ABB RAPID module: StanTargets.mod

MODULE StanTargets

	!Workplan Variables
	CONST string workplanName := "Stan";
	CONST string workplanUUID := "d4fdb9e9-5a3f-4a80-8776-aeeac0a44db1";

	!Workingsteps
	CONST string WorkPlan{20,6} := [
		["1","7", "Drilling.2", "b062b09d-c75e-4509-b058-f533fc3121cb", "Hole.101", "7ba2387a-5122-471d-9e62-f4dd978dd916"],
		["8","14", "Drilling.19", "bc6d7e2e-2011-44a2-96ea-1bdf43305bb2", "Hole.2", "a5a2d4b3-bce9-4376-9a01-39ac46aa03b7"],
		["15","21", "Drilling.20", "1d99434e-626c-49cd-aa28-89c40de30f06", "Hole.105", "77f1627f-4d66-488f-b970-3b2b6af52deb"],
		["22","28", "Drilling.3", "45a28ad3-0738-4ba8-bc95-27ca5d3c2a9d", "Hole.102", "83a55789-a548-457f-bc7a-c5f73e279b59"],
		["29","35", "Drilling.1", "9e701cf1-a52e-421d-a5d1-a7fe2dbaa640", "Hole.100", "ec9e4cb9-16a2-432e-8136-2d658a3c3d31"],
		["36","42", "Drilling.18", "90b44a9d-16c4-4a88-bf09-b7f65aff8308", "Hole.106", "8309f7bd-9ba6-4400-9e0b-e392acc79543"],
		["43","49", "Drilling.4", "301b61b0-be88-4471-af20-9d54f270abc0", "Hole.103", "543c12c8-ac8b-46e2-b23c-ed2f3937359b"],
		["50","56", "Drilling.17", "4a6a49de-cb15-4803-8bb7-097c767e5d1a", "Hole.107", "bc5d4dfc-6aa2-4544-8bb1-6cd32004e75e"],
		["57","63", "Drilling.21", "d6a29b26-5ed6-4fc9-a609-95bc5c10512a", "Hole.109", "c5793a88-d117-412a-8380-89480e2aa149"],
		["64","70", "Drilling.22", "32b13ef1-a017-413c-926d-f3ce9280a815", "Hole.110", "f43400ad-c29f-4157-ba87-1fd86718dbb4"],
		["71","77", "Drilling.23", "961958d8-0134-4891-910a-03c3b0fd50ac", "Hole.111", "4c4ae24f-0e25-46c1-affc-8b190d84e835"],
		["78","84", "Drilling.24", "46b8f9da-afaf-476f-bebf-76b29446400a", "Hole.112", "58a054b0-4018-4bcc-8be0-6224a9ae077a"],
		["85","91", "Drilling.37", "a26de890-fc0a-49b5-bfdf-50d0ba577d7f", "Hole.117", "fd2c949e-3c41-489a-8a46-dd0d10567b1b"],
		["92","98", "Drilling.38", "57e6c193-12b5-426e-af89-bc1afa04e779", "Hole.116", "13521d27-8989-4ee6-aa90-747ab0996569"],
		["99","105", "Drilling.39", "43fec44c-5451-4481-a3ed-f2154e5b5857", "Hole.115", "b8ea09e7-7ee5-4781-9867-97bdf0c7c8c2"],
		["106","112", "Drilling.40", "b2407ed9-3760-41ef-9af3-e4b017b94bad", "Hole.114", "6fd1afc0-306a-4e0e-985a-70eb87f380a3"],
		["113","119", "Drilling.41", "e4391847-02d9-4746-a9c4-e995e37bf0a5", "Hole.119", "2fe5694b-30b9-4983-885c-0907e4daf0a7"],
		["120","126", "Drilling.42", "9648c8b5-7603-4606-8e84-4fa243c23e6f", "Hole.120", "7e69786d-15ab-4ddf-bc4f-041c788858b9"],
		["127","133", "Drilling.43", "1797812d-a7bf-4001-89eb-f8bf3d30d00a", "Hole.121", "a39c1e68-904f-4878-9c68-b76c3ab1c433"],
		["134","140", "Drilling.44", "c9657693-5bc7-40ba-995c-70b253dd4bce", "Hole.122", "35b9f3e4-dbe9-4a3b-b0cd-96909b64c764"]
		];

	!Positions
	CONST robtarget WorkingstepRobtargets{140} := [
		[[289.186156636195,-206.403560128169,35.3771625636731],[0.00835255338347923,-0.000732758938354189,-0.996138888459216,-0.0873900040940131],[0,0,0,0],[9E+09,9E+09,9E+09,9E+09,9E+09,9E+09]],
		[[288.347319864636,-197.55839601017,-14.6398287952277],[0.00835255338347923,-0.000732758938354189,-0.996138888459216,-0.0873900040940131],[0,0,0,0],[9E+09,9E+09,9E+09,9E+09,9E+09,9E+09]],
		[[288.347319864636,-197.55839601017,-14.6398287952277],[0.00835255338347923,-0.000732758938354189,-0.996138888459216,-0.0873900040940131],[0,0,0,0],[9E+09,9E+09,9E+09,9E+09,9E+09,9E+09]],
		[[287.823046882412,-192.030168436421,-45.9004483945406],[0.00835255338347923,-0.000732758938354189,-0.996138888459216,-0.0873900040940131],[0,0,0,0],[9E+09,9E+09,9E+09,9E+09,9E+09,9E+09]],
		[[287.823046882412,-192.030168436421,-45.9004483945406],[0.00835255338347923,-0.000732758938354189,-0.996138888459216,-0.0873900040940131],[0,0,0,0],[9E+09,9E+09,9E+09,9E+09,9E+09,9E+09]],
		[[288.347319864636,-197.55839601017,-14.6398287952277],[0.00835255338347923,-0.000732758938354189,-0.996138888459216,-0.0873900040940131],[0,0,0,0],[9E+09,9E+09,9E+09,9E+09,9E+09,9E+09]],
		[[289.186156636195,-206.403560128169,35.3771625636731],[0.00835255338347923,-0.000732758938354189,-0.996138888459216,-0.0873900040940131],[0,0,0,0],[9E+09,9E+09,9E+09,9E+09,9E+09,9E+09]],
		[[254.909208192728,-190.980764818536,38.5531834909307],[0.00803255668836741,-0.000646350507138514,-0.996745854533864,-0.0802044994599877],[0,0,0,0],[9E+09,9E+09,9E+09,9E+09,9E+09,9E+09]],
		[[254.101023132797,-182.857977487938,-11.5866924850904],[0.00803255668836741,-0.000646350507138514,-0.996745854533864,-0.0802044994599877],[0,0,0,0],[9E+09,9E+09,9E+09,9E+09,9E+09,9E+09]],
		[[254.101023132797,-182.857977487938,-11.5866924850904],[0.00803255668836741,-0.000646350507138514,-0.996745854533864,-0.0802044994599877],[0,0,0,0],[9E+09,9E+09,9E+09,9E+09,9E+09,9E+09]],
		[[253.595907470339,-177.781235406315,-42.9241149701038],[0.00803255668836741,-0.000646350507138514,-0.996745854533864,-0.0802044994599877],[0,0,0,0],[9E+09,9E+09,9E+09,9E+09,9E+09,9E+09]],
		[[253.595907470339,-177.781235406315,-42.9241149701038],[0.00803255668836741,-0.000646350507138514,-0.996745854533864,-0.0802044994599877],[0,0,0,0],[9E+09,9E+09,9E+09,9E+09,9E+09,9E+09]],
		[[254.101023132797,-182.857977487938,-11.5866924850904],[0.00803255668836741,-0.000646350507138514,-0.996745854533864,-0.0802044994599877],[0,0,0,0],[9E+09,9E+09,9E+09,9E+09,9E+09,9E+09]],
		[[254.909208192728,-190.980764818536,38.5531834909307],[0.00803255668836741,-0.000646350507138514,-0.996745854533864,-0.0802044994599877],[0,0,0,0],[9E+09,9E+09,9E+09,9E+09,9E+09,9E+09]],
		[[255.049346094491,-251.794133959213,27.0746013914174],[0.00931771731230624,-0.000993284320775785,-0.994322356952738,-0.105996433875385],[0,0,0,0],[9E+09,9E+09,9E+09,9E+09,9E+09,9E+09]],
		[[254.118737842067,-241.085099842443,-22.5750769214012],[0.00931771731230624,-0.000993284320775785,-0.994322356952738,-0.105996433875385],[0,0,0,0],[9E+09,9E+09,9E+09,9E+09,9E+09,9E+09]],
		[[254.118737842067,-241.085099842443,-22.5750769214012],[0.00931771731230624,-0.000993284320775785,-0.994322356952738,-0.105996433875385],[0,0,0,0],[9E+09,9E+09,9E+09,9E+09,9E+09,9E+09]],
		[[253.5371076843,-234.391953519461,-53.6061258669128],[0.00931771731230624,-0.000993284320775785,-0.994322356952738,-0.105996433875385],[0,0,0,0],[9E+09,9E+09,9E+09,9E+09,9E+09,9E+09]],
		[[253.5371076843,-234.391953519461,-53.6061258669128],[0.00931771731230624,-0.000993284320775785,-0.994322356952738,-0.105996433875385],[0,0,0,0],[9E+09,9E+09,9E+09,9E+09,9E+09,9E+09]],
		[[254.118737842067,-241.085099842443,-22.5750769214012],[0.00931771731230624,-0.000993284320775785,-0.994322356952738,-0.105996433875385],[0,0,0,0],[9E+09,9E+09,9E+09,9E+09,9E+09,9E+09]],
		[[255.049346094491,-251.794133959213,27.0746013914174],[0.00931771731230624,-0.000993284320775785,-0.994322356952738,-0.105996433875385],[0,0,0,0],[9E+09,9E+09,9E+09,9E+09,9E+09,9E+09]],
		[[288.817292795415,-151.336810998548,43.7919561194079],[0.00741254609803812,-0.000475090293762373,-0.997924837913392,-0.0639597242417948],[0,0,0,0],[9E+09,9E+09,9E+09,9E+09,9E+09,9E+09]],
		[[288.068828229942,-144.851630260459,-6.58683139665437],[0.00741254609803812,-0.000475090293762373,-0.997924837913392,-0.0639597242417948],[0,0,0,0],[9E+09,9E+09,9E+09,9E+09,9E+09,9E+09]],
		[[288.068828229942,-144.851630260459,-6.58683139665437],[0.00741254609803812,-0.000475090293762373,-0.997924837913392,-0.0639597242417948],[0,0,0,0],[9E+09,9E+09,9E+09,9E+09,9E+09,9E+09]],
		[[287.60103787652,-140.798392299153,-38.0735735941933],[0.00741254609803812,-0.000475090293762373,-0.997924837913392,-0.0639597242417948],[0,0,0,0],[9E+09,9E+09,9E+09,9E+09,9E+09,9E+09]],
		[[287.60103787652,-140.798392299153,-38.0735735941933],[0.00741254609803812,-0.000475090293762373,-0.997924837913392,-0.0639597242417948],[0,0,0,0],[9E+09,9E+09,9E+09,9E+09,9E+09,9E+09]],
		[[288.068828229942,-144.851630260459,-6.58683139665437],[0.00741254609803812,-0.000475090293762373,-0.997924837913392,-0.0639597242417948],[0,0,0,0],[9E+09,9E+09,9E+09,9E+09,9E+09,9E+09]],
		[[288.817292795415,-151.336810998548,43.7919561194079],[0.00741254609803812,-0.000475090293762373,-0.997924837913392,-0.0639597242417948],[0,0,0,0],[9E+09,9E+09,9E+09,9E+09,9E+09,9E+09]],
		[[293.28700751171,-244.361649311658,27.9483297927613],[0.00918827288987244,-0.000958205797942005,-0.994563756282914,-0.103718813005981],[0,0,0,0],[9E+09,9E+09,9E+09,9E+09,9E+09,9E+09]],
		[[292.368651285828,-233.880209617552,-21.7501213277837],[0.00918827288987244,-0.000958205797942005,-0.994563756282914,-0.103718813005981],[0,0,0,0],[9E+09,9E+09,9E+09,9E+09,9E+09,9E+09]],
		[[292.368651285828,-233.880209617552,-21.7501213277837],[0.00918827288987244,-0.000958205797942005,-0.994563756282914,-0.103718813005981],[0,0,0,0],[9E+09,9E+09,9E+09,9E+09,9E+09,9E+09]],
		[[291.794678644652,-227.329309808736,-52.8116532781243],[0.00918827288987244,-0.000958205797942005,-0.994563756282914,-0.103718813005981],[0,0,0,0],[9E+09,9E+09,9E+09,9E+09,9E+09,9E+09]],
		[[291.794678644652,-227.329309808736,-52.8116532781243],[0.00918827288987244,-0.000958205797942005,-0.994563756282914,-0.103718813005981],[0,0,0,0],[9E+09,9E+09,9E+09,9E+09,9E+09,9E+09]],
		[[292.368651285828,-233.880209617552,-21.7501213277837],[0.00918827288987244,-0.000958205797942005,-0.994563756282914,-0.103718813005981],[0,0,0,0],[9E+09,9E+09,9E+09,9E+09,9E+09,9E+09]],
		[[293.28700751171,-244.361649311658,27.9483297927613],[0.00918827288987244,-0.000958205797942005,-0.994563756282914,-0.103718813005981],[0,0,0,0],[9E+09,9E+09,9E+09,9E+09,9E+09,9E+09]],
		[[249.459094617476,-137.316682571751,46.0807019976294],[0.00720641123076419,-0.000415118187492874,-0.998318997016837,-0.0575071778942388],[0,0,0,0],[9E+09,9E+09,9E+09,9E+09,9E+09,9E+09]],
		[[248.730579441892,-131.483471005379,-4.37802280255641],[0.00720641123076419,-0.000415118187492874,-0.998318997016837,-0.0575071778942388],[0,0,0,0],[9E+09,9E+09,9E+09,9E+09,9E+09,9E+09]],
		[[248.730579441892,-131.483471005379,-4.37802280255641],[0.00720641123076419,-0.000415118187492874,-0.998318997016837,-0.0575071778942388],[0,0,0,0],[9E+09,9E+09,9E+09,9E+09,9E+09,9E+09]],
		[[248.275257457153,-127.837713776397,-35.9147258026727],[0.00720641123076419,-0.000415118187492874,-0.998318997016837,-0.0575071778942388],[0,0,0,0],[9E+09,9E+09,9E+09,9E+09,9E+09,9E+09]],
		[[248.275257457153,-127.837713776397,-35.9147258026727],[0.00720641123076419,-0.000415118187492874,-0.998318997016837,-0.0575071778942388],[0,0,0,0],[9E+09,9E+09,9E+09,9E+09,9E+09,9E+09]],
		[[248.730579441892,-131.483471005379,-4.37802280255641],[0.00720641123076419,-0.000415118187492874,-0.998318997016837,-0.0575071778942388],[0,0,0,0],[9E+09,9E+09,9E+09,9E+09,9E+09,9E+09]],
		[[249.459094617476,-137.316682571751,46.0807019976294],[0.00720641123076419,-0.000415118187492874,-0.998318997016837,-0.0575071778942388],[0,0,0,0],[9E+09,9E+09,9E+09,9E+09,9E+09,9E+09]],
		[[290.829543745998,-100.056182181525,49.234722450473],[0.00680707504627507,-0.000287946923608445,-0.999083317268074,-0.042262346982922],[0,0,0,0],[9E+09,9E+09,9E+09,9E+09,9E+09,9E+09]],
		[[290.139815300174,-95.7660646865366,-1.37910141761904],[0.00680707504627507,-0.000287946923608445,-0.999083317268074,-0.042262346982922],[0,0,0,0],[9E+09,9E+09,9E+09,9E+09,9E+09,9E+09]],
		[[290.139815300174,-95.7660646865366,-1.37910141761904],[0.00680707504627507,-0.000287946923608445,-0.999083317268074,-0.042262346982922],[0,0,0,0],[9E+09,9E+09,9E+09,9E+09,9E+09,9E+09]],
		[[289.708735021536,-93.0847412521693,-33.0127413351765],[0.00680707504627507,-0.000287946923608445,-0.999083317268074,-0.042262346982922],[0,0,0,0],[9E+09,9E+09,9E+09,9E+09,9E+09,9E+09]],
		[[289.708735021536,-93.0847412521693,-33.0127413351765],[0.00680707504627507,-0.000287946923608445,-0.999083317268074,-0.042262346982922],[0,0,0,0],[9E+09,9E+09,9E+09,9E+09,9E+09,9E+09]],
		[[290.139815300174,-95.7660646865366,-1.37910141761904],[0.00680707504627507,-0.000287946923608445,-0.999083317268074,-0.042262346982922],[0,0,0,0],[9E+09,9E+09,9E+09,9E+09,9E+09,9E+09]],
		[[290.829543745998,-100.056182181525,49.234722450473],[0.00680707504627507,-0.000287946923608445,-0.999083317268074,-0.042262346982922],[0,0,0,0],[9E+09,9E+09,9E+09,9E+09,9E+09,9E+09]],
		[[245.740187119161,-87.6128069534354,50.8276032034953],[0.0066909782554097,-0.000245268224154555,-0.999306424862602,-0.0366311326852939],[0,0,0,0],[9E+09,9E+09,9E+09,9E+09,9E+09,9E+09]],
		[[245.061768043552,-83.8934984330366,0.16848268519243],[0.0066909782554097,-0.000245268224154555,-0.999306424862602,-0.0366311326852939],[0,0,0,0],[9E+09,9E+09,9E+09,9E+09,9E+09,9E+09]],
		[[245.061768043552,-83.8934984330366,0.16848268519243],[0.0066909782554097,-0.000245268224154555,-0.999306424862602,-0.0366311326852939],[0,0,0,0],[9E+09,9E+09,9E+09,9E+09,9E+09,9E+09]],
		[[244.637756121297,-81.5689306077871,-31.493467638747],[0.0066909782554097,-0.000245268224154555,-0.999306424862602,-0.0366311326852939],[0,0,0,0],[9E+09,9E+09,9E+09,9E+09,9E+09,9E+09]],
		[[244.637756121297,-81.5689306077871,-31.493467638747],[0.0066909782554097,-0.000245268224154555,-0.999306424862602,-0.0366311326852939],[0,0,0,0],[9E+09,9E+09,9E+09,9E+09,9E+09,9E+09]],
		[[245.061768043552,-83.8934984330366,0.16848268519243],[0.0066909782554097,-0.000245268224154555,-0.999306424862602,-0.0366311326852939],[0,0,0,0],[9E+09,9E+09,9E+09,9E+09,9E+09,9E+09]],
		[[245.740187119161,-87.6128069534354,50.8276032034953],[0.0066909782554097,-0.000245268224154555,-0.999306424862602,-0.0366311326852939],[0,0,0,0],[9E+09,9E+09,9E+09,9E+09,9E+09,9E+09]],
		[[403.099233829671,-245.749127372575,25.6017542319324],[0.00936954043940217,-0.00100794170503457,-0.994219250722917,-0.106954556973674],[0,0,0,0],[9E+09,9E+09,9E+09,9E+09,9E+09,9E+09]],
		[[402.163744360367,-234.944401870427,-24.0270959086467],[0.00936954043940217,-0.00100794170503457,-0.994219250722917,-0.106954556973674],[0,0,0,0],[9E+09,9E+09,9E+09,9E+09,9E+09,9E+09]],
		[[402.163744360367,-234.944401870427,-24.0270959086467],[0.00936954043940217,-0.00100794170503457,-0.994219250722917,-0.106954556973674],[0,0,0,0],[9E+09,9E+09,9E+09,9E+09,9E+09,9E+09]],
		[[401.579063442052,-228.191448431585,-55.0451272465088],[0.00936954043940217,-0.00100794170503457,-0.994219250722917,-0.106954556973674],[0,0,0,0],[9E+09,9E+09,9E+09,9E+09,9E+09,9E+09]],
		[[401.579063442052,-228.191448431585,-55.0451272465088],[0.00936954043940217,-0.00100794170503457,-0.994219250722917,-0.106954556973674],[0,0,0,0],[9E+09,9E+09,9E+09,9E+09,9E+09,9E+09]],
		[[402.163744360367,-234.944401870427,-24.0270959086467],[0.00936954043940217,-0.00100794170503457,-0.994219250722917,-0.106954556973674],[0,0,0,0],[9E+09,9E+09,9E+09,9E+09,9E+09,9E+09]],
		[[403.099233829671,-245.749127372575,25.6017542319324],[0.00936954043940217,-0.00100794170503457,-0.994219250722917,-0.106954556973674],[0,0,0,0],[9E+09,9E+09,9E+09,9E+09,9E+09,9E+09]],
		[[396.033748937128,-194.18703812988,35.7216135201404],[0.00820516010917249,-0.000693329099167655,-0.996415168384063,-0.0841962401565701],[0,0,0,0],[9E+09,9E+09,9E+09,9E+09,9E+09,9E+09]],
		[[395.209024115822,-185.662788001459,-14.3513031985533],[0.00820516010917249,-0.000693329099167655,-0.996415168384063,-0.0841962401565701],[0,0,0,0],[9E+09,9E+09,9E+09,9E+09,9E+09,9E+09]],
		[[395.209024115822,-185.662788001459,-14.3513031985533],[0.00820516010917249,-0.000693329099167655,-0.996415168384063,-0.0841962401565701],[0,0,0,0],[9E+09,9E+09,9E+09,9E+09,9E+09,9E+09]],
		[[394.693571102503,-180.335131671196,-45.6468761477369],[0.00820516010917249,-0.000693329099167655,-0.996415168384063,-0.0841962401565701],[0,0,0,0],[9E+09,9E+09,9E+09,9E+09,9E+09,9E+09]],
		[[394.693571102503,-180.335131671196,-45.6468761477369],[0.00820516010917249,-0.000693329099167655,-0.996415168384063,-0.0841962401565701],[0,0,0,0],[9E+09,9E+09,9E+09,9E+09,9E+09,9E+09]],
		[[395.209024115822,-185.662788001459,-14.3513031985533],[0.00820516010917249,-0.000693329099167655,-0.996415168384063,-0.0841962401565701],[0,0,0,0],[9E+09,9E+09,9E+09,9E+09,9E+09,9E+09]],
		[[396.033748937128,-194.18703812988,35.7216135201404],[0.00820516010917249,-0.000693329099167655,-0.996415168384063,-0.0841962401565701],[0,0,0,0],[9E+09,9E+09,9E+09,9E+09,9E+09,9E+09]],
		[[391.06989532529,-137.544241837855,44.000996564666],[0.00726571628808549,-0.000432828028158066,-0.998203897421597,-0.0594642850714026],[0,0,0,0],[9E+09,9E+09,9E+09,9E+09,9E+09,9E+09]],
		[[390.335639388971,-131.51320224425,-6.43438218517918],[0.00726571628808549,-0.000432828028158066,-0.998203897421597,-0.0594642850714026],[0,0,0,0],[9E+09,9E+09,9E+09,9E+09,9E+09,9E+09]],
		[[390.335639388971,-131.51320224425,-6.43438218517918],[0.00726571628808549,-0.000432828028158066,-0.998203897421597,-0.0594642850714026],[0,0,0,0],[9E+09,9E+09,9E+09,9E+09,9E+09,9E+09]],
		[[389.876729428771,-127.743802498246,-37.9564939038324],[0.00726571628808549,-0.000432828028158066,-0.998203897421597,-0.0594642850714026],[0,0,0,0],[9E+09,9E+09,9E+09,9E+09,9E+09,9E+09]],
		[[389.876729428771,-127.743802498246,-37.9564939038324],[0.00726571628808549,-0.000432828028158066,-0.998203897421597,-0.0594642850714026],[0,0,0,0],[9E+09,9E+09,9E+09,9E+09,9E+09,9E+09]],
		[[390.335639388971,-131.51320224425,-6.43438218517918],[0.00726571628808549,-0.000432828028158066,-0.998203897421597,-0.0594642850714026],[0,0,0,0],[9E+09,9E+09,9E+09,9E+09,9E+09,9E+09]],
		[[391.06989532529,-137.544241837855,44.000996564666],[0.00726571628808549,-0.000432828028158066,-0.998203897421597,-0.0594642850714026],[0,0,0,0],[9E+09,9E+09,9E+09,9E+09,9E+09,9E+09]],
		[[385.668546901666,-85.4729115296458,49.1107245728777],[0.00669526575096486,-0.000247046366600005,-0.999297509827073,-0.0368727438364299],[0,0,0,0],[9E+09,9E+09,9E+09,9E+09,9E+09,9E+09]],
		[[384.989711265164,-81.7291044236946,-1.54658576365773],[0.00669526575096486,-0.000247046366600005,-0.999297509827073,-0.0368727438364299],[0,0,0,0],[9E+09,9E+09,9E+09,9E+09,9E+09,9E+09]],
		[[384.989711265164,-81.7291044236946,-1.54658576365773],[0.00669526575096486,-0.000247046366600005,-0.999297509827073,-0.0368727438364299],[0,0,0,0],[9E+09,9E+09,9E+09,9E+09,9E+09,9E+09]],
		[[384.565438992351,-79.389224982475,-33.2074047239924],[0.00669526575096486,-0.000247046366600005,-0.999297509827073,-0.0368727438364299],[0,0,0,0],[9E+09,9E+09,9E+09,9E+09,9E+09,9E+09]],
		[[384.565438992351,-79.389224982475,-33.2074047239924],[0.00669526575096486,-0.000247046366600005,-0.999297509827073,-0.0368727438364299],[0,0,0,0],[9E+09,9E+09,9E+09,9E+09,9E+09,9E+09]],
		[[384.989711265164,-81.7291044236946,-1.54658576365773],[0.00669526575096486,-0.000247046366600005,-0.999297509827073,-0.0368727438364299],[0,0,0,0],[9E+09,9E+09,9E+09,9E+09,9E+09,9E+09]],
		[[385.668546901666,-85.4729115296458,49.1107245728777],[0.00669526575096486,-0.000247046366600005,-0.999297509827073,-0.0368727438364299],[0,0,0,0],[9E+09,9E+09,9E+09,9E+09,9E+09,9E+09]],
		[[478.315791276222,-86.4437658870823,47.794069485851],[0.00671892774812616,-0.000256146261682229,-0.999251517650421,-0.038094551740885],[0,0,0,0],[9E+09,9E+09,9E+09,9E+09,9E+09,9E+09]],
		[[477.634650553439,-82.5760815046593,-2.85390248572684],[0.00671892774812616,-0.000256146261682229,-0.999251517650421,-0.038094551740885],[0,0,0,0],[9E+09,9E+09,9E+09,9E+09,9E+09,9E+09]],
		[[477.634650553439,-82.5760815046593,-2.85390248572684],[0.00671892774812616,-0.000256146261682229,-0.999251517650421,-0.038094551740885],[0,0,0,0],[9E+09,9E+09,9E+09,9E+09,9E+09,9E+09]],
		[[477.208937601699,-80.1587787656448,-34.5088849679627],[0.00671892774812616,-0.000256146261682229,-0.999251517650421,-0.038094551740885],[0,0,0,0],[9E+09,9E+09,9E+09,9E+09,9E+09,9E+09]],
		[[477.208937601699,-80.1587787656448,-34.5088849679627],[0.00671892774812616,-0.000256146261682229,-0.999251517650421,-0.038094551740885],[0,0,0,0],[9E+09,9E+09,9E+09,9E+09,9E+09,9E+09]],
		[[477.634650553439,-82.5760815046593,-2.85390248572684],[0.00671892774812616,-0.000256146261682229,-0.999251517650421,-0.038094551740885],[0,0,0,0],[9E+09,9E+09,9E+09,9E+09,9E+09,9E+09]],
		[[478.315791276222,-86.4437658870823,47.794069485851],[0.00671892774812616,-0.000256146261682229,-0.999251517650421,-0.038094551740885],[0,0,0,0],[9E+09,9E+09,9E+09,9E+09,9E+09,9E+09]],
		[[483.133106013849,-138.756801668918,42.5082331765351],[0.0073226084519266,-0.000449565472182051,-0.998093827794076,-0.0612771426856401],[0,0,0,0],[9E+09,9E+09,9E+09,9E+09,9E+09,9E+09]],
		[[482.393346029146,-132.54257687196,-7.904822328343],[0.0073226084519266,-0.000449565472182051,-0.998093827794076,-0.0612771426856401],[0,0,0,0],[9E+09,9E+09,9E+09,9E+09,9E+09,9E+09]],
		[[482.393346029146,-132.54257687196,-7.904822328343],[0.0073226084519266,-0.000449565472182051,-0.998093827794076,-0.0612771426856401],[0,0,0,0],[9E+09,9E+09,9E+09,9E+09,9E+09,9E+09]],
		[[481.930996038707,-128.658686373861,-39.4129820188915],[0.0073226084519266,-0.000449565472182051,-0.998093827794076,-0.0612771426856401],[0,0,0,0],[9E+09,9E+09,9E+09,9E+09,9E+09,9E+09]],
		[[481.930996038707,-128.658686373861,-39.4129820188915],[0.0073226084519266,-0.000449565472182051,-0.998093827794076,-0.0612771426856401],[0,0,0,0],[9E+09,9E+09,9E+09,9E+09,9E+09,9E+09]],
		[[482.393346029146,-132.54257687196,-7.904822328343],[0.0073226084519266,-0.000449565472182051,-0.998093827794076,-0.0612771426856401],[0,0,0,0],[9E+09,9E+09,9E+09,9E+09,9E+09,9E+09]],
		[[483.133106013849,-138.756801668918,42.5082331765351],[0.0073226084519266,-0.000449565472182051,-0.998093827794076,-0.0612771426856401],[0,0,0,0],[9E+09,9E+09,9E+09,9E+09,9E+09,9E+09]],
		[[483.222642292122,-189.861338067738,35.0219683114554],[0.00819448846874309,-0.000690679339774657,-0.996433068445667,-0.0839851976763621],[0,0,0,0],[9E+09,9E+09,9E+09,9E+09,9E+09,9E+09]],
		[[482.39894544337,-181.3583032081,-15.0545723206324],[0.00819448846874309,-0.000690679339774657,-0.996433068445667,-0.0839851976763621],[0,0,0,0],[9E+09,9E+09,9E+09,9E+09,9E+09,9E+09]],
		[[482.39894544337,-181.3583032081,-15.0545723206324],[0.00819448846874309,-0.000690679339774657,-0.996433068445667,-0.0839851976763621],[0,0,0,0],[9E+09,9E+09,9E+09,9E+09,9E+09,9E+09]],
		[[481.884134912899,-176.043906420827,-46.3524102156873],[0.00819448846874309,-0.000690679339774657,-0.996433068445667,-0.0839851976763621],[0,0,0,0],[9E+09,9E+09,9E+09,9E+09,9E+09,9E+09]],
		[[481.884134912899,-176.043906420827,-46.3524102156873],[0.00819448846874309,-0.000690679339774657,-0.996433068445667,-0.0839851976763621],[0,0,0,0],[9E+09,9E+09,9E+09,9E+09,9E+09,9E+09]],
		[[482.39894544337,-181.3583032081,-15.0545723206324],[0.00819448846874309,-0.000690679339774657,-0.996433068445667,-0.0839851976763621],[0,0,0,0],[9E+09,9E+09,9E+09,9E+09,9E+09,9E+09]],
		[[483.222642292122,-189.861338067738,35.0219683114554],[0.00819448846874309,-0.000690679339774657,-0.996433068445667,-0.0839851976763621],[0,0,0,0],[9E+09,9E+09,9E+09,9E+09,9E+09,9E+09]],
		[[489.630453604917,-244.907439108101,24.1464954374401],[0.00947203461223947,-0.00103629582389185,-0.994023250292104,-0.108751940350465],[0,0,0,0],[9E+09,9E+09,9E+09,9E+09,9E+09,9E+09]],
		[[488.685296902346,-233.923282965952,-25.4427674392399],[0.00947203461223947,-0.00103629582389185,-0.994023250292104,-0.108751940350465],[0,0,0,0],[9E+09,9E+09,9E+09,9E+09,9E+09,9E+09]],
		[[488.685296902346,-233.923282965952,-25.4427674392399],[0.00947203461223947,-0.00103629582389185,-0.994023250292104,-0.108751940350465],[0,0,0,0],[9E+09,9E+09,9E+09,9E+09,9E+09,9E+09]],
		[[488.094573963238,-227.058185377108,-56.4360567371645],[0.00947203461223947,-0.00103629582389185,-0.994023250292104,-0.108751940350465],[0,0,0,0],[9E+09,9E+09,9E+09,9E+09,9E+09,9E+09]],
		[[488.094573963238,-227.058185377108,-56.4360567371645],[0.00947203461223947,-0.00103629582389185,-0.994023250292104,-0.108751940350465],[0,0,0,0],[9E+09,9E+09,9E+09,9E+09,9E+09,9E+09]],
		[[488.685296902346,-233.923282965952,-25.4427674392399],[0.00947203461223947,-0.00103629582389185,-0.994023250292104,-0.108751940350465],[0,0,0,0],[9E+09,9E+09,9E+09,9E+09,9E+09,9E+09]],
		[[489.630453604917,-244.907439108101,24.1464954374401],[0.00947203461223947,-0.00103629582389185,-0.994023250292104,-0.108751940350465],[0,0,0,0],[9E+09,9E+09,9E+09,9E+09,9E+09,9E+09]],
		[[602.136376955429,-240.655233611394,22.9421139308661],[0.00952750400653266,-0.0010519700999858,-0.993913882382944,-0.109742035851254],[0,0,0,0],[9E+09,9E+09,9E+09,9E+09,9E+09,9E+09]],
		[[601.186003122767,-229.572283406206,-26.6250627521719],[0.00952750400653266,-0.0010519700999858,-0.993913882382944,-0.109742035851254],[0,0,0,0],[9E+09,9E+09,9E+09,9E+09,9E+09,9E+09]],
		[[601.186003122767,-229.572283406206,-26.6250627521719],[0.00952750400653266,-0.0010519700999858,-0.993913882382944,-0.109742035851254],[0,0,0,0],[9E+09,9E+09,9E+09,9E+09,9E+09,9E+09]],
		[[600.592019477353,-222.645439527964,-57.604548179071],[0.00952750400653266,-0.0010519700999858,-0.993913882382944,-0.109742035851254],[0,0,0,0],[9E+09,9E+09,9E+09,9E+09,9E+09,9E+09]],
		[[600.592019477353,-222.645439527964,-57.604548179071],[0.00952750400653266,-0.0010519700999858,-0.993913882382944,-0.109742035851254],[0,0,0,0],[9E+09,9E+09,9E+09,9E+09,9E+09,9E+09]],
		[[601.186003122767,-229.572283406206,-26.6250627521719],[0.00952750400653266,-0.0010519700999858,-0.993913882382944,-0.109742035851254],[0,0,0,0],[9E+09,9E+09,9E+09,9E+09,9E+09,9E+09]],
		[[602.136376955429,-240.655233611394,22.9421139308661],[0.00952750400653266,-0.0010519700999858,-0.993913882382944,-0.109742035851254],[0,0,0,0],[9E+09,9E+09,9E+09,9E+09,9E+09,9E+09]],
		[[594.105058195658,-186.41205556819,33.7829943400776],[0.00822215146796232,-0.000698454025213563,-0.996377418391712,-0.0846401116863593],[0,0,0,0],[9E+09,9E+09,9E+09,9E+09,9E+09,9E+09]],
		[[593.278720114878,-177.843188909236,-16.2822799481687],[0.00822215146796232,-0.000698454025213563,-0.996377418391712,-0.0846401116863593],[0,0,0,0],[9E+09,9E+09,9E+09,9E+09,9E+09,9E+09]],
		[[593.278720114878,-177.843188909236,-16.2822799481687],[0.00822215146796232,-0.000698454025213563,-0.996377418391712,-0.0846401116863593],[0,0,0,0],[9E+09,9E+09,9E+09,9E+09,9E+09,9E+09]],
		[[592.762258814391,-172.48764724739,-47.5730763783227],[0.00822215146796232,-0.000698454025213563,-0.996377418391712,-0.0846401116863593],[0,0,0,0],[9E+09,9E+09,9E+09,9E+09,9E+09,9E+09]],
		[[592.762258814391,-172.48764724739,-47.5730763783227],[0.00822215146796232,-0.000698454025213563,-0.996377418391712,-0.0846401116863593],[0,0,0,0],[9E+09,9E+09,9E+09,9E+09,9E+09,9E+09]],
		[[593.278720114878,-177.843188909236,-16.2822799481687],[0.00822215146796232,-0.000698454025213563,-0.996377418391712,-0.0846401116863593],[0,0,0,0],[9E+09,9E+09,9E+09,9E+09,9E+09,9E+09]],
		[[594.105058195658,-186.41205556819,33.7829943400776],[0.00822215146796232,-0.000698454025213563,-0.996377418391712,-0.0846401116863593],[0,0,0,0],[9E+09,9E+09,9E+09,9E+09,9E+09,9E+09]],
		[[594.013579836482,-136.119059315104,41.2060164577616],[0.00733540540573417,-0.000453473807444863,-0.99806765566097,-0.0617004125792975],[0,0,0,0],[9E+09,9E+09,9E+09,9E+09,9E+09,9E+09]],
		[[593.272585498753,-129.862072839968,-9.20173143521038],[0.00733540540573417,-0.000453473807444863,-0.99806765566097,-0.0617004125792975],[0,0,0,0],[9E+09,9E+09,9E+09,9E+09,9E+09,9E+09]],
		[[593.272585498753,-129.862072839968,-9.20173143521038],[0.00733540540573417,-0.000453473807444863,-0.99806765566097,-0.0617004125792975],[0,0,0,0],[9E+09,9E+09,9E+09,9E+09,9E+09,9E+09]],
		[[592.809464037672,-125.951456293008,-40.7065738683178],[0.00733540540573417,-0.000453473807444863,-0.99806765566097,-0.0617004125792975],[0,0,0,0],[9E+09,9E+09,9E+09,9E+09,9E+09,9E+09]],
		[[592.809464037672,-125.951456293008,-40.7065738683178],[0.00733540540573417,-0.000453473807444863,-0.99806765566097,-0.0617004125792975],[0,0,0,0],[9E+09,9E+09,9E+09,9E+09,9E+09,9E+09]],
		[[593.272585498753,-129.862072839968,-9.20173143521038],[0.00733540540573417,-0.000453473807444863,-0.99806765566097,-0.0617004125792975],[0,0,0,0],[9E+09,9E+09,9E+09,9E+09,9E+09,9E+09]],
		[[594.013579836482,-136.119059315104,41.2060164577616],[0.00733540540573417,-0.000453473807444863,-0.99806765566097,-0.0617004125792975],[0,0,0,0],[9E+09,9E+09,9E+09,9E+09,9E+09,9E+09]],
		[[593.951420595743,-86.0463664067457,46.2676477594915],[0.00673606385428096,-0.000262673005791383,-0.999217855075423,-0.0389645293198063],[0,0,0,0],[9E+09,9E+09,9E+09,9E+09,9E+09,9E+09]],
		[[593.268611664579,-82.090486810967,-4.37348955581023],[0.00673606385428096,-0.000262673005791383,-0.999217855075423,-0.0389645293198063],[0,0,0,0],[9E+09,9E+09,9E+09,9E+09,9E+09,9E+09]],
		[[593.268611664579,-82.090486810967,-4.37348955581023],[0.00673606385428096,-0.000262673005791383,-0.999217855075423,-0.0389645293198063],[0,0,0,0],[9E+09,9E+09,9E+09,9E+09,9E+09,9E+09]],
		[[592.841856082603,-79.6180620636052,-36.0242003778737],[0.00673606385428096,-0.000262673005791383,-0.999217855075423,-0.0389645293198063],[0,0,0,0],[9E+09,9E+09,9E+09,9E+09,9E+09,9E+09]],
		[[592.841856082603,-79.6180620636052,-36.0242003778737],[0.00673606385428096,-0.000262673005791383,-0.999217855075423,-0.0389645293198063],[0,0,0,0],[9E+09,9E+09,9E+09,9E+09,9E+09,9E+09]],
		[[593.268611664579,-82.090486810967,-4.37348955581023],[0.00673606385428096,-0.000262673005791383,-0.999217855075423,-0.0389645293198063],[0,0,0,0],[9E+09,9E+09,9E+09,9E+09,9E+09,9E+09]],
		[[593.951420595743,-86.0463664067457,46.2676477594915],[0.00673606385428096,-0.000262673005791383,-0.999217855075423,-0.0389645293198063],[0,0,0,0],[9E+09,9E+09,9E+09,9E+09,9E+09,9E+09]]
		];

	!Speeds
	CONST speeddata WorkingstepSpeeddatas{140} := [
		[ 800, 500, 5000, 1000],
		[ 800, 500, 5000, 1000],
		[ 4.23333333333333, 500, 5000, 1000],
		[ 4.23333333333333, 500, 5000, 1000],
		[ 800, 500, 5000, 1000],
		[ 800, 500, 5000, 1000],
		[ 800, 500, 5000, 1000],
		[ 800, 500, 5000, 1000],
		[ 800, 500, 5000, 1000],
		[ 4.23333333333333, 500, 5000, 1000],
		[ 4.23333333333333, 500, 5000, 1000],
		[ 800, 500, 5000, 1000],
		[ 800, 500, 5000, 1000],
		[ 800, 500, 5000, 1000],
		[ 800, 500, 5000, 1000],
		[ 800, 500, 5000, 1000],
		[ 4.23333333333333, 500, 5000, 1000],
		[ 4.23333333333333, 500, 5000, 1000],
		[ 800, 500, 5000, 1000],
		[ 800, 500, 5000, 1000],
		[ 800, 500, 5000, 1000],
		[ 800, 500, 5000, 1000],
		[ 800, 500, 5000, 1000],
		[ 4.23333333333333, 500, 5000, 1000],
		[ 4.23333333333333, 500, 5000, 1000],
		[ 800, 500, 5000, 1000],
		[ 800, 500, 5000, 1000],
		[ 800, 500, 5000, 1000],
		[ 800, 500, 5000, 1000],
		[ 800, 500, 5000, 1000],
		[ 4.23333333333333, 500, 5000, 1000],
		[ 4.23333333333333, 500, 5000, 1000],
		[ 800, 500, 5000, 1000],
		[ 800, 500, 5000, 1000],
		[ 800, 500, 5000, 1000],
		[ 800, 500, 5000, 1000],
		[ 800, 500, 5000, 1000],
		[ 4.23333333333333, 500, 5000, 1000],
		[ 4.23333333333333, 500, 5000, 1000],
		[ 800, 500, 5000, 1000],
		[ 800, 500, 5000, 1000],
		[ 800, 500, 5000, 1000],
		[ 800, 500, 5000, 1000],
		[ 800, 500, 5000, 1000],
		[ 4.23333333333333, 500, 5000, 1000],
		[ 4.23333333333333, 500, 5000, 1000],
		[ 800, 500, 5000, 1000],
		[ 800, 500, 5000, 1000],
		[ 800, 500, 5000, 1000],
		[ 800, 500, 5000, 1000],
		[ 800, 500, 5000, 1000],
		[ 4.23333333333333, 500, 5000, 1000],
		[ 4.23333333333333, 500, 5000, 1000],
		[ 800, 500, 5000, 1000],
		[ 800, 500, 5000, 1000],
		[ 800, 500, 5000, 1000],
		[ 800, 500, 5000, 1000],
		[ 800, 500, 5000, 1000],
		[ 4.23333333333333, 500, 5000, 1000],
		[ 4.23333333333333, 500, 5000, 1000],
		[ 800, 500, 5000, 1000],
		[ 800, 500, 5000, 1000],
		[ 800, 500, 5000, 1000],
		[ 800, 500, 5000, 1000],
		[ 800, 500, 5000, 1000],
		[ 4.23333333333333, 500, 5000, 1000],
		[ 4.23333333333333, 500, 5000, 1000],
		[ 800, 500, 5000, 1000],
		[ 800, 500, 5000, 1000],
		[ 800, 500, 5000, 1000],
		[ 800, 500, 5000, 1000],
		[ 800, 500, 5000, 1000],
		[ 4.23333333333333, 500, 5000, 1000],
		[ 4.23333333333333, 500, 5000, 1000],
		[ 800, 500, 5000, 1000],
		[ 800, 500, 5000, 1000],
		[ 800, 500, 5000, 1000],
		[ 800, 500, 5000, 1000],
		[ 800, 500, 5000, 1000],
		[ 4.23333333333333, 500, 5000, 1000],
		[ 4.23333333333333, 500, 5000, 1000],
		[ 800, 500, 5000, 1000],
		[ 800, 500, 5000, 1000],
		[ 800, 500, 5000, 1000],
		[ 800, 500, 5000, 1000],
		[ 800, 500, 5000, 1000],
		[ 4.23333333333333, 500, 5000, 1000],
		[ 4.23333333333333, 500, 5000, 1000],
		[ 800, 500, 5000, 1000],
		[ 800, 500, 5000, 1000],
		[ 800, 500, 5000, 1000],
		[ 800, 500, 5000, 1000],
		[ 800, 500, 5000, 1000],
		[ 4.23333333333333, 500, 5000, 1000],
		[ 4.23333333333333, 500, 5000, 1000],
		[ 800, 500, 5000, 1000],
		[ 800, 500, 5000, 1000],
		[ 800, 500, 5000, 1000],
		[ 800, 500, 5000, 1000],
		[ 800, 500, 5000, 1000],
		[ 4.23333333333333, 500, 5000, 1000],
		[ 4.23333333333333, 500, 5000, 1000],
		[ 800, 500, 5000, 1000],
		[ 800, 500, 5000, 1000],
		[ 800, 500, 5000, 1000],
		[ 800, 500, 5000, 1000],
		[ 800, 500, 5000, 1000],
		[ 4.23333333333333, 500, 5000, 1000],
		[ 4.23333333333333, 500, 5000, 1000],
		[ 800, 500, 5000, 1000],
		[ 800, 500, 5000, 1000],
		[ 800, 500, 5000, 1000],
		[ 800, 500, 5000, 1000],
		[ 800, 500, 5000, 1000],
		[ 4.23333333333333, 500, 5000, 1000],
		[ 4.23333333333333, 500, 5000, 1000],
		[ 800, 500, 5000, 1000],
		[ 800, 500, 5000, 1000],
		[ 800, 500, 5000, 1000],
		[ 800, 500, 5000, 1000],
		[ 800, 500, 5000, 1000],
		[ 4.23333333333333, 500, 5000, 1000],
		[ 4.23333333333333, 500, 5000, 1000],
		[ 800, 500, 5000, 1000],
		[ 800, 500, 5000, 1000],
		[ 800, 500, 5000, 1000],
		[ 800, 500, 5000, 1000],
		[ 800, 500, 5000, 1000],
		[ 4.23333333333333, 500, 5000, 1000],
		[ 4.23333333333333, 500, 5000, 1000],
		[ 800, 500, 5000, 1000],
		[ 800, 500, 5000, 1000],
		[ 800, 500, 5000, 1000],
		[ 800, 500, 5000, 1000],
		[ 800, 500, 5000, 1000],
		[ 4.23333333333333, 500, 5000, 1000],
		[ 4.23333333333333, 500, 5000, 1000],
		[ 800, 500, 5000, 1000],
		[ 800, 500, 5000, 1000],
		[ 800, 500, 5000, 1000]
		];


ENDMODULE
